// TIA Portal project "Siemens PLC" (V21)

(* hardware
DEVICE "ET 200SP station_1"  ET 200SP-Station
   slot 0: "Rack_0"  Rack  6ES5 710-8MAx1
   slot 1: "PLC_1"  CPU 1510SP-1 PN  6ES7 510-1DK03-0AB0  V4.1
      slot 32768: "PROFINET interface_1"  X1
         slot 32771: "Port_3"  X1 P3
   slot 2: "Server module_1"  Server module  6ES7 193-6PA00-0AA0  V1.2
      slot 1: "Server module_1"  Server module
   slot 127: "BA 2xRJ45"  BA 2xRJ45  6ES7 193-6AR00-0AA0  V0.0
      slot 32769: "Port_1"  X1 P1  6ES7 193-6AR00-0AA0
      slot 32770: "Port_2"  X1 P2  6ES7 193-6AR00-0AA0
*)

// ===== PLC "PLC_1"  CPU 1510SP-1 PN =====

VAR_GLOBAL   // PLC tag table "Default tag table"
   "System_Byte" AT %MB1 : Byte;
   "FirstScan" AT %M1.0 : Bool;
   "DiagStatusUpdate" AT %M1.1 : Bool;
   "AlwaysTRUE" AT %M1.2 : Bool;
   "AlwaysFALSE" AT %M1.3 : Bool;
   "Clock_Byte" AT %MB0 : Byte;
   "Clock_10Hz" AT %M0.0 : Bool;
   "Clock_5Hz" AT %M0.1 : Bool;
   "Clock_2.5Hz" AT %M0.2 : Bool;
   "Clock_2Hz" AT %M0.3 : Bool;
   "Clock_1.25Hz" AT %M0.4 : Bool;
   "Clock_1Hz" AT %M0.5 : Bool;
   "Clock_0.625Hz" AT %M0.6 : Bool;
   "Clock_0.5Hz" AT %M0.7 : Bool;
END_VAR

TYPE "Data"
   STRUCT
      sDateTime : String;
      iVar : Int;
      xVar : Bool;
      idVar : DInt;
      flVar : Real;
   END_STRUCT;
END_TYPE

DATA_BLOCK "DB_Optimized"   // DB1
{ S7_Optimized_Access := 'TRUE' }
VERSION : 0.1
BEGIN
END_DATA_BLOCK

DATA_BLOCK "DB_NonOptimized"   // DB2
{ S7_Optimized_Access := 'FALSE' }
VERSION : 0.1
BEGIN
END_DATA_BLOCK

DATA_BLOCK "SimulateData_DB"   // DB3
{ S7_Optimized_Access := 'TRUE' }
VERSION : 0.1
// stored: InstanceOfName SimulateData
"SimulateData"
BEGIN
END_DATA_BLOCK

FUNCTION_BLOCK "SimulateData"   // FB1, LAD
{ S7_Optimized_Access := 'TRUE' }
VERSION : 0.1
   VAR
      CurrDTL : DTL;
   END_VAR
   VAR_TEMP
      tmpInt : Int;
      tmpMin : Real;
      tmpSec : Real;
      tmpNanoSec : Real;
   END_VAR
BEGIN

REGION Network 1: Get current time
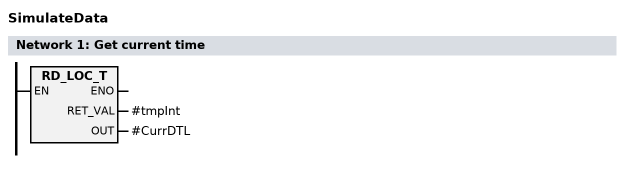
   #tmpInt := RD_LOC_T(OUT => #CurrDTL);
END_REGION

REGION Network 2 (SCL): Convert dtl to string
   "DB_Optimized".sDateTime := CONCAT(IN1:=DELETE(IN:=UINT_TO_STRING(#CurrDTL.YEAR), L := 1, P := 1),
                                      IN2:='-',
                                      IN3:=DELETE(IN:=USINT_TO_STRING(#CurrDTL.MONTH), L := 1, P := 1),
                                      IN4:='-',
                                      IN5:=DELETE(IN:=USINT_TO_STRING(#CurrDTL.DAY), L := 1, P := 1),
                                      IN6:=' - ',
                                      IN7:=DELETE(IN:=USINT_TO_STRING(#CurrDTL.HOUR), L := 1, P := 1),
                                      IN8:=':',
                                      IN9:=DELETE(IN:=USINT_TO_STRING(#CurrDTL.MINUTE), L := 1, P := 1),
                                      IN10:=':',
                                      IN11:=DELETE(IN:=USINT_TO_STRING(#CurrDTL.SECOND), L := 1, P := 1));
END_REGION

REGION Network 3 (SCL): Move simple simulation variables
   "DB_Optimized".iVar := #CurrDTL.SECOND;
   "DB_Optimized".xVar := "Clock_10Hz";
   "DB_Optimized".idVar := UDINT_TO_DINT(#CurrDTL.NANOSECOND);
END_REGION

REGION Network 4 (SCL): Randon variable
   #tmpMin := USINT_TO_REAL(#CurrDTL.MINUTE);
   #tmpSec := USINT_TO_REAL(#CurrDTL.SECOND);
   #tmpNanoSec := UDINT_TO_REAL(#CurrDTL.NANOSECOND) / 100000;

   IF (#tmpSec <> 0) AND (#tmpMin <> 0) THEN
       "DB_Optimized".flVar := (#tmpNanoSec / #tmpSec + #tmpNanoSec / #tmpMin) / #tmpSec;
   ELSE
       #tmpSec := 100;
       #tmpMin := 200;
       "DB_Optimized".flVar := (#tmpNanoSec / #tmpSec + #tmpNanoSec / #tmpMin) / #tmpSec;
   END_IF;

   // Avoid NaN number
   IF "DB_Optimized".flVar <> "DB_Optimized".flVar THEN
       "DB_Optimized".flVar := 0;
   END_IF;
END_REGION
END_FUNCTION_BLOCK

ORGANIZATION_BLOCK "Main"   // OB1, LAD, ProgramCycle
TITLE = "Main Program Sweep (Cycle)"
{ S7_Optimized_Access := 'TRUE' }
VERSION : 0.1
   VAR_INPUT
      Initial_Call : Bool;   // Initial call of this OB
      Remanence : Bool;   // =True, if remanent data are available
   END_VAR
BEGIN

REGION Network 1
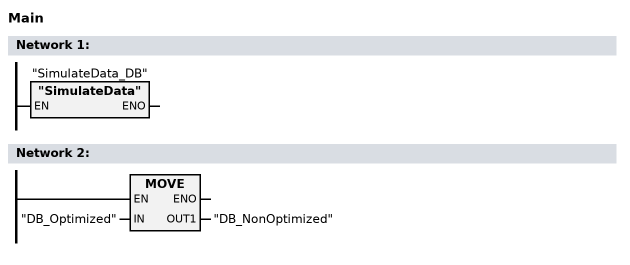
   RUNG wire#powerrail
      "SimulateData_DB"()
   END_RUNG
   // the same network as SCL:
   "SimulateData_DB"();   // "SimulateData"
END_REGION

REGION Network 2
   RUNG wire#powerrail
      Move(in := "DB_Optimized", out1 => "DB_NonOptimized")
   END_RUNG
   // the same network as SCL:
   "DB_NonOptimized" := "DB_Optimized";
END_REGION
END_ORGANIZATION_BLOCK